Yaskawa INFORM job: KRIS1A_HARDOX.JBI

/JOB
//NAME KRIS1A_HARDOX
//POS
///NPOS 114,114,112,5,0,0
///TOOL 0
///POSTYPE PULSE
///PULSE
C00000=15349,-87390,-111573,-674,86554,-86826
C00001=-110984,-87390,-111570,-673,86559,8331
C00002=-111759,-79535,-69021,-454,64406,8169
C00003=-114095,-78681,-67160,402,63698,7299
C00004=-114095,-78325,-65957,403,63140,7298
C00005=-114095,-78648,-67045,402,63644,7299
C00006=-113114,-93112,-73015,43,59884,7664
C00007=-114174,-91151,-70215,449,59172,7253
C00008=-114269,-89568,-69588,484,59599,7218
C00009=-112804,-96361,-75693,-76,59862,7786
C00010=-111133,-79411,-68712,-683,64284,8404
C00011=-110795,-77497,-66452,-807,63881,8532
C00012=-110795,-77213,-65470,-810,63423,8535
C00013=-111147,-78773,-67027,-680,63577,8402
C00014=-109795,-94038,-73387,-1221,59664,8950
C00015=-110034,-90449,-69592,-1136,59169,8863
C00016=-110197,-88771,-68919,-1070,59614,8797
C00017=-109724,-95740,-76085,-1239,60450,8969
C00018=-97790,-93891,-80845,-5517,64828,13352
C00019=-95102,58941,36484,-30043,98742,46310
C00020=-95139,59332,36927,-30037,98667,46316
C00021=-123036,27157,-10763,-19283,86742,21526
C00022=-150798,39984,8064,-10438,77055,13413
C00023=-150701,50951,18953,-20501,80603,7648
C00024=-146523,55066,28554,-32677,81611,-991
C00025=-149211,60857,35994,-32225,79233,-1370
C00026=-149329,62991,38450,-32233,78844,-1300
C00027=-150515,78276,52468,-28887,85234,-3452
C00028=-150515,78429,53961,-28913,84496,-3266
C00029=-149211,60857,35994,-32225,79233,-1370
C00030=-141139,35393,-539,-16647,85388,2500
C00031=-139001,60609,30102,-17411,80166,3961
C00032=-135441,52818,21854,-13680,80270,7361
C00033=-135777,54342,23766,-13597,79830,7293
C00034=-135983,57253,27023,-13543,79305,7282
C00035=-135093,72210,41659,-15118,85737,6681
C00036=-135093,72171,42757,-15126,85066,6764
C00037=-135777,54342,23766,-13597,79830,7293
C00038=-130802,76085,44553,-22242,86386,17390
C00039=-130308,68928,40049,-22014,82627,18301
C00040=-129747,65534,38183,-22158,82221,18578
C00041=-131607,88324,51934,-23272,94341,15485
C00042=-139696,65014,36490,-20940,85073,14420
C00043=-150319,81140,52112,-36023,87083,-4429
C00044=-147546,82233,57744,-41634,87908,-4895
C00045=-133755,47291,19718,-43086,89514,541
C00046=-130254,27624,-12420,-14523,95031,2735
C00047=-123724,-37006,-66316,-16306,84508,85949
C00048=-116979,-69120,-74771,-25636,74961,89025
C00049=-117994,-43372,-61454,-24127,91092,85341
C00050=-149498,-32155,-54450,-17063,84771,75512
C00051=-141330,-38704,-51094,-33432,76685,78426
C00052=-130528,-69811,-74379,-36386,79670,81887
C00053=-132947,-100822,-92962,-36380,74991,82451
C00054=15349,-87390,-111573,-674,86554,-86826
C00055=15349,-87390,-111573,-674,86554,-86826
C00056=15349,-87390,-111570,-674,86556,-86825
C00057=3643,-76224,-106676,19950,71810,76872
C00058=15349,-87390,-111570,-674,86556,-86825
C00059=-68824,-87390,-111568,-659,86557,2288
C00060=-102324,-63179,-76492,-4543,93838,9300
C00061=-99268,-62121,-71685,-4896,91607,10397
C00062=-101449,-61888,-70084,-4627,90618,9708
C00063=-101449,-61917,-69079,-4627,89987,9729
C00064=-101449,-61887,-70112,-4627,90636,9704
C00065=-98771,-79826,-78849,-4944,86964,10742
C00066=-97205,-87840,-78173,-7148,76765,11690
C00067=-97422,-86698,-77695,-7095,77039,11596
C00068=-98458,-92698,-83162,-6885,77230,11227
C00069=-70334,-47845,-62333,-11740,90555,19804
C00070=-68889,-44293,-58067,-11955,89977,20346
C00071=-68889,-44364,-57255,-11953,89453,20397
C00072=-68889,-44289,-58112,-11958,90008,20343
C00073=-63676,-56068,-65467,-12713,89294,22180
C00074=-64287,-54843,-62333,-12625,87932,22111
C00075=-64982,-53370,-61506,-12527,88068,21862
C00076=-63556,-56320,-65366,-12731,89128,22240
C00077=-105066,-71099,-78115,-5454,84680,8612
C00078=-112264,29903,-5613,20852,82012,58
C00079=-116025,40020,6760,22161,80694,-1490
C00080=-115757,40485,7245,22080,80570,-1418
C00081=-116380,72893,34300,23392,97175,1652
C00082=-116380,72712,34934,23360,96730,1564
C00083=-113337,19398,-6828,21452,77926,-1043
C00084=-112260,2825,-16849,21290,75457,-1102
C00085=-114727,-25650,-50489,21683,81747,-843
C00086=-114727,-25650,-50489,21683,81747,-843
C00087=-78893,324,-30560,8500,76378,10543
C00088=-78852,1478,-33213,8418,78578,10708
C00089=-79073,11671,-16805,8667,73792,10299
C00090=-79033,12633,-15939,8651,73747,10311
C00091=-81241,30994,-8525,12450,88846,11360
C00092=-81241,30688,-7880,12449,88305,11306
C00093=-79073,11131,-13779,8761,71676,10146
C00094=-92259,55371,29296,14706,84689,187
C00095=-93263,53762,27321,13271,84592,849
C00096=-96212,48835,21669,8946,83923,2815
C00097=-101108,42280,16538,-5466,77936,-2086
C00098=-101169,55733,34354,-23908,75396,-5221
C00099=-101120,57575,40115,-31807,71578,-5564
C00100=-101198,55593,39781,-34332,69056,-5141
C00101=-99101,24615,5399,-28066,67939,-3113
C00102=-101092,-2809,-21504,5594,61806,151
C00103=-116279,-103565,-87668,15153,52841,-6820
C00104=-136626,-108292,-100051,23905,62636,71559
C00105=-181552,-118218,-82845,46514,74578,55658
C00106=-187474,-110161,-80368,46081,79459,55112
C00107=-145536,-97007,-88996,9555,84002,75248
C00108=-145251,-96121,-85437,9544,82257,75216
C00109=-99167,-97649,-86024,2499,78276,90872
C00110=-118631,-91766,-78858,25217,81137,84835
C00111=-117699,-93504,-86004,20553,84337,85672
C00112=-134531,-91540,-85241,22037,89209,80450
C00113=3161,-91504,-85468,2682,88050,79011
BC00000=115,663699,1075117
BC00001=171753,674879,306456
BC00002=55475,735323,199167
BC00003=55475,735323,199167
BC00004=55475,735323,199167
BC00005=55475,735323,199167
BC00006=55475,735323,199167
BC00007=55475,735323,199167
BC00008=55475,735323,199167
BC00009=55475,735323,199167
BC00010=108320,735323,199167
BC00011=108320,735323,199167
BC00012=108320,735323,199167
BC00013=108320,735323,199167
BC00014=108320,735323,199167
BC00015=108320,735323,199167
BC00016=108320,735323,199167
BC00017=108320,735323,199167
BC00018=108320,735323,199167
BC00019=108320,749563,199167
BC00020=108320,749563,199167
BC00021=153902,806828,124230
BC00022=190527,806828,124230
BC00023=190527,806828,124230
BC00024=190527,806828,124230
BC00025=190526,806828,124220
BC00026=190526,806828,124219
BC00027=190526,806828,124219
BC00028=190526,806828,124219
BC00029=190526,806828,124220
BC00030=190527,806828,124230
BC00031=190527,806828,124230
BC00032=170092,806828,124230
BC00033=170092,806828,124230
BC00034=170092,806828,124229
BC00035=170092,806828,124229
BC00036=170092,806828,124229
BC00037=170092,806828,124230
BC00038=172528,806828,89212
BC00039=170093,806828,124227
BC00040=170093,806828,124227
BC00041=170093,806828,47158
BC00042=170093,806828,124224
BC00043=193689,806828,68198
BC00044=185222,806828,81006
BC00045=170093,806828,124227
BC00046=170093,806828,124227
BC00047=170093,806828,124227
BC00048=170093,743154,124227
BC00049=170093,743154,124227
BC00050=170093,743154,124227
BC00051=170093,743154,124227
BC00052=170093,743154,124227
BC00053=170093,743154,124227
BC00054=115,663699,1075117
BC00055=115,663699,1075117
BC00056=115,663700,1075116
BC00057=199464,674570,1075173
BC00058=141263,687330,337717
BC00059=222435,751088,164876
BC00060=279925,751088,164876
BC00061=279925,751088,164876
BC00062=279925,751088,164876
BC00063=279925,751088,164876
BC00064=279925,751088,164876
BC00065=279925,751088,164876
BC00066=279925,751088,164876
BC00067=279925,751088,164876
BC00068=279925,751088,164876
BC00069=279925,751088,164876
BC00070=279925,751088,164876
BC00071=279925,751088,164876
BC00072=279925,751088,164876
BC00073=279925,751088,164876
BC00074=279925,751088,164876
BC00075=279925,751088,164876
BC00076=279925,751088,164876
BC00077=279925,751088,164876
BC00078=279925,819641,96131
BC00079=292926,813604,89674
BC00080=292926,813604,89674
BC00081=292926,813604,66237
BC00082=292926,813604,66237
BC00083=286680,834738,133855
BC00084=279925,834738,164876
BC00085=279925,834738,164876
BC00086=279925,762190,164876
BC00087=244896,762190,164876
BC00088=278481,826600,115077
BC00089=278481,826600,115468
BC00090=278481,826600,115468
BC00091=278481,826600,82693
BC00092=278481,826600,82693
BC00093=278481,826600,138122
BC00094=302666,794256,164873
BC00095=305731,794256,164873
BC00096=314980,794256,164873
BC00097=326440,794256,164872
BC00098=326440,794254,164870
BC00099=326440,794256,164871
BC00100=326440,794256,164873
BC00101=326440,794256,164873
BC00102=326440,794256,164873
BC00103=326440,794256,164873
BC00104=326440,794256,164873
BC00105=326885,794948,164297
BC00106=326885,794948,164297
BC00107=326885,794948,164297
BC00108=326885,794948,164297
BC00109=326885,794948,164297
BC00110=326885,794948,164295
BC00111=326885,794948,164295
BC00112=326885,737668,213736
BC00113=87842,675035,1040975
EC00000=798157,0
EC00001=798154,2
EC00002=798154,2
EC00003=798154,2
EC00004=798154,2
EC00005=798154,2
EC00006=798154,2
EC00007=798154,2
EC00008=798154,2
EC00009=798154,2
EC00010=798154,2
EC00011=798154,2
EC00012=798154,2
EC00013=798154,2
EC00014=798154,2
EC00015=798154,2
EC00016=798154,2
EC00017=798154,2
EC00018=798154,2
EC00019=798154,2
EC00020=798154,2
EC00021=798154,2
EC00022=798154,2
EC00023=798154,2
EC00024=798154,2
EC00025=798150,3
EC00026=798134,12
EC00027=798134,12
EC00028=798134,12
EC00029=798150,3
EC00030=798154,2
EC00031=798154,2
EC00032=798154,2
EC00033=798154,2
EC00034=798153,3
EC00035=798153,3
EC00036=798153,3
EC00037=798154,2
EC00038=798153,2
EC00039=798151,3
EC00040=798151,3
EC00041=798141,9
EC00042=798150,3
EC00043=798153,2
EC00044=798153,2
EC00045=798153,2
EC00046=798153,2
EC00047=798153,2
EC00048=798153,2
EC00049=798153,2
EC00050=798153,2
EC00051=798153,2
EC00052=798157,0
EC00053=93266,10480
EC00054=184298,1105644
EC00055=798157,1112952
EC00056=798157,1112952
EC00057=798156,1112951
EC00058=798156,1112951
EC00059=798156,1112951
EC00060=798156,1112951
EC00061=798156,1112951
EC00062=798156,1112951
EC00063=798156,1112951
EC00064=798156,1112951
EC00065=798156,1112951
EC00066=798156,1112951
EC00067=798156,1112951
EC00068=798156,1112951
EC00069=798156,1112951
EC00070=798156,1112951
EC00071=798156,1112951
EC00072=798156,1112951
EC00073=798156,1112951
EC00074=798156,1112951
EC00075=798156,1112951
EC00076=798156,1112951
EC00077=798156,1112951
EC00078=798156,1112951
EC00079=798156,1112951
EC00080=798156,1112951
EC00081=798156,1112951
EC00082=798156,1112951
EC00083=798156,1112951
EC00084=798156,1112951
EC00085=798156,1112951
EC00086=798156,1112951
EC00087=798156,1112951
EC00088=798156,1112951
EC00089=798156,1112951
EC00090=798156,1112951
EC00091=798156,1112951
EC00092=798155,1112950
EC00093=798155,1112950
EC00094=798155,1112950
EC00095=798154,1112949
EC00096=798153,1112949
EC00097=798154,1112949
EC00098=798155,1112950
EC00099=798155,1112950
EC00100=798155,1112950
EC00101=798155,1112950
EC00102=798155,1112950
EC00103=798155,1112950
EC00104=798155,1112950
EC00105=798155,1112950
EC00106=798155,1112950
EC00107=798155,1112950
EC00108=798154,1112948
EC00109=798154,1112948
EC00110=798154,1112948
EC00111=798154,1103372
///POSTYPE BASE
///RECTAN
///RCONF 0,0,0,0,0,0,0,0,0,0,0,0,0,0,0,0,0,0,0,0,0,0,0,0
P00006=0.222,-3.123,-1.508,0.0000,0.0000,0.0000
P00021=-0.225,-6.128,-0.405,0.0000,0.0000,0.0000
P00022=0.222,-3.123,-1.508,0.0000,0.0000,0.0000
P00023=0.143,-0.036,0.682,0.0000,0.0000,0.0000
P00024=0.145,-0.552,1.326,0.0000,0.0000,0.0000
//INST
///DATE 2025/01/21 10:54
///ATTR SC,RW
///GROUP1 RB1,BS1
///GROUP2 ST1
NOP
CALL JOB:CLEAN-R1_KM_3P
MOVJ C00000 BC00000 VJ=100.00  +MOVJ EC00000 VJ=100.00
MOVJ C00001 BC00001 VJ=100.00  +MOVJ EC00001 VJ=100.00
MOVJ C00002 BC00002 VJ=100.00  +MOVJ EC00002 VJ=100.00
SMOVL C00003 BC00003 V=100.0  +MOVJ EC00003
SREFP 3 C00004 BC00004  +REFP EC00004
CALL JOB:SEARCH-R1-S13D
SET P023 P006
SFTON3D P023
SMOVL C00005 BC00005 V=133.3  +MOVJ EC00005
SMOVL C00006 BC00006 V=133.3  +MOVJ EC00006
SMOVL C00007 BC00007 V=133.3  +MOVJ EC00007
SREFP 3 C00008 BC00008  +REFP EC00008
CALL JOB:SEARCH-R1-S13D
SET P023 P006
SFTON3D P023
SMOVL C00009 BC00009 V=166.7  +MOVJ EC00009
SFTOF3D
SMOVL C00010 BC00010 V=250.0  +MOVJ EC00010
SMOVL C00011 BC00011 V=100.0  +MOVJ EC00011
SREFP 3 C00012 BC00012  +REFP EC00012
CALL JOB:SEARCH-R1-S13D
SET P024 P006
SFTON3D P024
SMOVL C00013 BC00013 V=133.3  +MOVJ EC00013
SMOVL C00014 BC00014 V=133.3  +MOVJ EC00014
SMOVL C00015 BC00015 V=133.3  +MOVJ EC00015
SREFP 3 C00016 BC00016  +REFP EC00016
CALL JOB:SEARCH-R1-S13D
SET P024 P006
SFTON3D P024
SMOVL C00017 BC00017 V=166.7  +MOVJ EC00017
SFTOF3D
MOVJ C00018 BC00018 VJ=100.00  +MOVJ EC00018 VJ=100.00
SMOVL C00019 BC00019 V=500.0  +MOVJ EC00019
MOVJ C00020 BC00020 VJ=100.00  +MOVJ EC00020 VJ=100.00
MOVJ C00021 BC00021 VJ=100.00  +MOVJ EC00021 VJ=20.00
MOVJ C00022 BC00022 VJ=20.00  +MOVJ EC00022 VJ=20.00
MOVJ C00023 BC00023 VJ=20.00  +MOVJ EC00023 VJ=20.00
MOVJ C00024 BC00024 VJ=20.00  +MOVJ EC00024 VJ=20.00
SMOVL C00025 BC00025 V=100.0  +MOVJ EC00025
SREFP 3 C00026 BC00026  +REFP EC00026
CALL JOB:SEARCH-R1-S13D
SET P022 P006
SFTON3D P022
SMOVL C00027 BC00027 V=100.0  +MOVJ EC00027
SREFP 3 C00028 BC00028  +REFP EC00028
CALL JOB:SEARCH-R1-S13D
SET P022 P006
SFTON3D P022
SMOVL C00029 BC00029 V=100.0  +MOVJ EC00029
SFTOF3D
MOVL C00030 BC00030 V=500.0  +MOVJ EC00030 VJ=20.00
MOVL C00031 BC00031 V=500.0  +MOVJ EC00031 VJ=20.00
SMOVL C00032 BC00032 V=500.0  +MOVJ EC00032
SMOVL C00033 BC00033 V=100.0  +MOVJ EC00033
SREFP 3 C00034 BC00034  +REFP EC00034
CALL JOB:SEARCH-R1-S13D
SET P021 P006
SFTON3D P021
SMOVL C00035 BC00035 V=100.0  +MOVJ EC00035
SREFP 3 C00036 BC00036  +REFP EC00036
CALL JOB:SEARCH-R1-S13D
SET P021 P006
SFTON3D P021
SMOVL C00037 BC00037 V=100.0  +MOVJ EC00037
MACRO1 MJ#(0) ARGF21
SMOVL C00038 BC00038 V=166.7 PL=0  +MOVJ EC00038
REFP 1 RB1 C00039 BC00039
REFP 2 RB1 C00040 BC00040
ARCON
SWVON WEV#(100)
SMOVL C00041 BC00041 V=8.3  +MOVJ EC00039
SFTON3D P022
SMOVL C00042 BC00042 V=8.3  +MOVJ EC00040
SMOVL C00043 BC00043 V=8.3  +MOVJ EC00041
SMOVL C00044 BC00044 V=8.3  +MOVJ EC00042
ARCOF
SWVOF
SFTOF3D
SMOVL C00045 BC00045 V=333.3  +MOVJ EC00043
SMOVL C00046 BC00046 V=666.7  +MOVJ EC00044
SMOVL C00047 BC00047 V=666.7  +MOVJ EC00045
SFTOF3D
SMOVL C00048 BC00048 V=333.3  +MOVJ EC00046
SFTON3D P024
SMOVL C00049 BC00049 V=166.7  +MOVJ EC00047
ARCON
SWVON WEV#(20)
SFTON3D P023
SMOVL C00050 BC00050 V=12.5  +MOVJ EC00048
SMOVL C00051 BC00051 V=12.5  +MOVJ EC00049
ARCOF
SWVOF
SFTOF3D
SMOVL C00052 BC00052 V=500.0  +MOVJ EC00050
SMOVL C00053 BC00053 V=1000.0  +MOVJ EC00051
MOVJ C00054 BC00054 VJ=100.00  +MOVJ EC00052 VJ=20.00
MOVJ C00055 BC00055 VJ=100.00  +MOVJ EC00053 VJ=100.00
MOVJ C00056 BC00056 VJ=100.00  +MOVJ EC00054 VJ=100.00
MOVJ C00057 BC00057 VJ=100.00  +MOVJ EC00055 VJ=100.00
'DRUGA STRONA
CALL JOB:CLEAN-R1_KM_3P
MOVJ C00058 BC00058 VJ=100.00  +MOVJ EC00056 VJ=100.00
MOVJ C00059 BC00059 VJ=100.00  +MOVJ EC00057 VJ=100.00
MOVJ C00060 BC00060 VJ=100.00  +MOVJ EC00058 VJ=100.00
MOVJ C00061 BC00061 VJ=100.00  +MOVJ EC00059 VJ=100.00
SMOVL C00062 BC00062 V=166.7  +MOVJ EC00060
SREFP 3 C00063 BC00063  +REFP EC00061
CALL JOB:SEARCH-R1-S13D
SET P023 P006
SFTON3D P023
SMOVL C00064 BC00064 V=250.0  +MOVJ EC00062
SMOVL C00065 BC00065 V=250.0  +MOVJ EC00063
SMOVL C00066 BC00066 V=250.0  +MOVJ EC00064
SREFP 3 C00067 BC00067  +REFP EC00065
CALL JOB:SEARCH-R1-S13D
SET P023 P006
SFTON3D P023
SFTOF3D
SMOVL C00068 BC00068 V=250.0  +MOVJ EC00066
SMOVL C00069 BC00069 V=250.0  +MOVJ EC00067
SMOVL C00070 BC00070 V=250.0  +MOVJ EC00068
SREFP 3 C00071 BC00071  +REFP EC00069
CALL JOB:SEARCH-R1-S13D
SET P024 P006
SFTON3D P024
SMOVL C00072 BC00072 V=250.0  +MOVJ EC00070
SMOVL C00073 BC00073 V=250.0  +MOVJ EC00071
SMOVL C00074 BC00074 V=250.0  +MOVJ EC00072
SREFP 3 C00075 BC00075  +REFP EC00073
CALL JOB:SEARCH-R1-S13D
SET P024 P006
SFTON3D P024
SFTOF3D
SMOVL C00076 BC00076 V=250.0  +MOVJ EC00074
MOVJ C00077 BC00077 VJ=100.00  +MOVJ EC00075 VJ=100.00
SMOVL C00078 BC00078 V=666.7  +MOVJ EC00076
SMOVL C00079 BC00079 V=250.0  +MOVJ EC00077
SREFP 3 C00080 BC00080  +REFP EC00078
CALL JOB:SEARCH-R1-S13D
SET P021 P006
SFTON3D P021
SMOVL C00081 BC00081 V=250.0  +MOVJ EC00079
SREFP 3 C00082 BC00082  +REFP EC00080
CALL JOB:SEARCH-R1-S13D
SET P021 P006
SFTON3D P021
SFTOF3D
SMOVL C00083 BC00083 V=250.0  +MOVJ EC00081
MOVL C00084 BC00084 V=250.0  +MOVJ EC00082 VJ=20.00
MOVL C00085 BC00085 V=333.3  +MOVJ EC00083 VJ=20.00
SMOVL C00086 BC00086 V=1000.0  +MOVJ EC00084
SMOVL C00087 BC00087 V=1000.0  +MOVJ EC00085
SMOVL C00088 BC00088 V=250.0  +MOVJ EC00086
SMOVL C00089 BC00089 V=250.0  +MOVJ EC00087
SREFP 3 C00090 BC00090  +REFP EC00088
CALL JOB:SEARCH-R1-S13D
SET P022 P006
SFTON3D P022
SMOVL C00091 BC00091 V=250.0  +MOVJ EC00089
SREFP 3 C00092 BC00092  +REFP EC00090
CALL JOB:SEARCH-R1-S13D
SET P022 P006
SFTON3D P022
SFTOF3D
SMOVL C00093 BC00093 V=250.0  +MOVJ EC00091
MACRO1 MJ#(0) ARGF21
SFTON3D P022
SMOVL C00094 BC00094 V=166.7 PL=0  +MOVJ EC00092
ARCON
SWVON WEV#(100)
SMOVL C00095 BC00095 V=8.3  +MOVJ EC00093
SMOVL C00096 BC00096 V=8.3  +MOVJ EC00094
SMOVL C00097 BC00097 V=8.3  +MOVJ EC00095
SFTON3D P021
SMOVL C00098 BC00098 V=8.3  +MOVJ EC00096
SMOVL C00099 BC00099 V=8.3  +MOVJ EC00097
SMOVL C00100 BC00100 V=8.3  +MOVJ EC00098
ARCOF
SWVOF
SMOVL C00101 BC00101 V=250.0  +MOVJ EC00099
SMOVL C00102 BC00102 V=500.0  +MOVJ EC00100
MOVJ C00103 BC00103 VJ=50.00  +MOVJ EC00101 VJ=20.00
MOVJ C00104 BC00104 VJ=100.00  +MOVJ EC00102 VJ=20.00
SMOVL C00105 BC00105 V=500.0  +MOVJ EC00103
SMOVL C00106 BC00106 V=250.0  +MOVJ EC00104
MOVL C00107 BC00107 V=250.0  +MOVJ EC00105 VJ=100.00
SFTON3D P023
SMOVL C00108 BC00108 V=250.0  +MOVJ EC00106
ARCON
SWVON WEV#(20)
SFTON3D P024
SMOVL C00109 BC00109 V=11.7  +MOVJ EC00107
SMOVL C00110 BC00110 V=11.7  +MOVJ EC00108
ARCOF
SWVOF
SFTOF3D
SMOVL C00111 BC00111 V=250.0  +MOVJ EC00109
MOVJ C00112 BC00112 VJ=100.00  +MOVJ EC00110 VJ=20.00
MOVJ C00113 BC00113 VJ=100.00  +MOVJ EC00111 VJ=100.00
END
